TYPE roboArmsRecipe :
STRUCT
	
	fixtureNum     : INT    := 48;                    // Брой сензори в тара
	waitPos24      : BOOL   := FALSE;                 // Чакащата позиция е HEX24
	waitPos27      : BOOL   := TRUE;                  // Чакащата позиция е HEX27
	rotAngle       : REAL   := 180.0;                 // Ъгъл на завъртане

END_STRUCT
END_TYPE

(* stored: Version 1.1.0.1, ProductVersion 3.1.4024.3
   DUT roboArmsRecipe: Id {92be77a0-ff3f-47b1-9b6c-71037a04ef8e} *)
